SYSTEM ASM_MVCDR (* Assembly System Control+Diagnostics+HMI with Remote Model+View *)
  (* Standard: 61499-1; Classification: Simulation; ApplicationDomain: Assembly; Type: Dual Stroke Cylinder *)
  (* Version 1.0, 2007-11-08, JHC, Holobloc Inc, Changed PRESS_ACT socket from 1027 to 1031. *)
  (* Version 0.9, 2007-07-07, JHC, Holobloc Inc, Added DIAGNOSTICS.LOG.RUN. *)
  (* Version 0.8, 2007-07-07, JHC, Holobloc Inc, Accelerated simulation, adjusted diagnostics; added ASM_GATE to TRANSPORT_MDL, PRESS_MDL. *)
  (* Version 0.7, 2007-07-06, JHC, Holobloc Inc, Simplified MODEL.CLOCK as in ASM_MVCDL. *)
  (* Version 0.6, 2007-07-06, JHC, Holobloc Inc, Added initial readout of TRANSPORT_ACT, PRESS_ACT. *)
  (* Version 0.5, 2007-07-06, JHC, Holobloc Inc, Adjusted order of resources so timing-sensitive initialization is always done last. *)
  (* Version 0.4, 2007-07-05, JHC, Holobloc Inc, Made device order MODEL, DIAGNOSTICS, CONTROL (startup is reverse order). *)
  (* Version 0.3, 2007-07-03, JHC, Holobloc Inc, Updated MODEL.CLOCK as in ASM_MVCL. *)
  (* Version 0.2, 2007-01-15, JHC, Holobloc Inc, Converted I/O to tagged data. *)
  (* Version 0.1, 2004-10-21, JHC, Rockwell Automation, Adapted to new Load/Unload model. *)
  (* Version 0.0, 2004-09-26, JHC, Rockwell Automation, Extended from ASM_MVCDL1. *)
  DEVICE MODEL : RMT_FRAME(BOUNDS := [380,100,185,160])
    RESOURCE MGR : RMT_RES
    END_RESOURCE
    RESOURCE CLOCK : EMB_RES
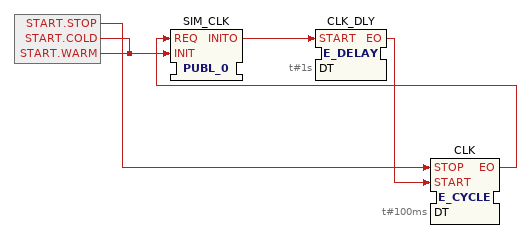
      FBS
        CLK : E_CYCLE(DT := t#100ms);
        SIM_CLK : PUBL_0;
        CLK_DLY : E_DELAY(DT := t#1s); (* Wait for everything to initialize, then start simulation *)
      END_FBS
      EVENT_CONNECTIONS
        CLK.EO TO SIM_CLK.REQ;
        START.STOP TO CLK.STOP;
        START.COLD TO SIM_CLK.INIT;
        START.WARM TO SIM_CLK.INIT;
        SIM_CLK.INITO TO CLK_DLY.START;
        CLK_DLY.EO TO CLK.START;
      END_CONNECTIONS
    END_RESOURCE
    RESOURCE TAGS : EMB_RES
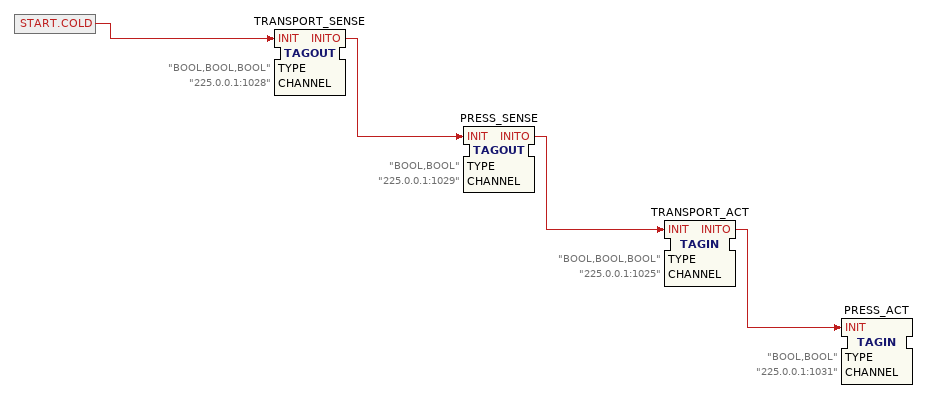
      FBS
        TRANSPORT_SENSE : TAGOUT(TYPE := "BOOL,BOOL,BOOL", CHANNEL := "225.0.0.1:1028");
        TRANSPORT_ACT : TAGIN(TYPE := "BOOL,BOOL,BOOL", CHANNEL := "225.0.0.1:1025");
        PRESS_SENSE : TAGOUT(TYPE := "BOOL,BOOL", CHANNEL := "225.0.0.1:1029");
        PRESS_ACT : TAGIN(TYPE := "BOOL,BOOL", CHANNEL := "225.0.0.1:1031");
      END_FBS
      EVENT_CONNECTIONS
        START.COLD TO TRANSPORT_SENSE.INIT;
        TRANSPORT_ACT.INITO TO PRESS_ACT.INIT;
        TRANSPORT_SENSE.INITO TO PRESS_SENSE.INIT;
        PRESS_SENSE.INITO TO TRANSPORT_ACT.INIT;
      END_CONNECTIONS
    END_RESOURCE
    RESOURCE TRANSPORT_MDL : EMB_RES
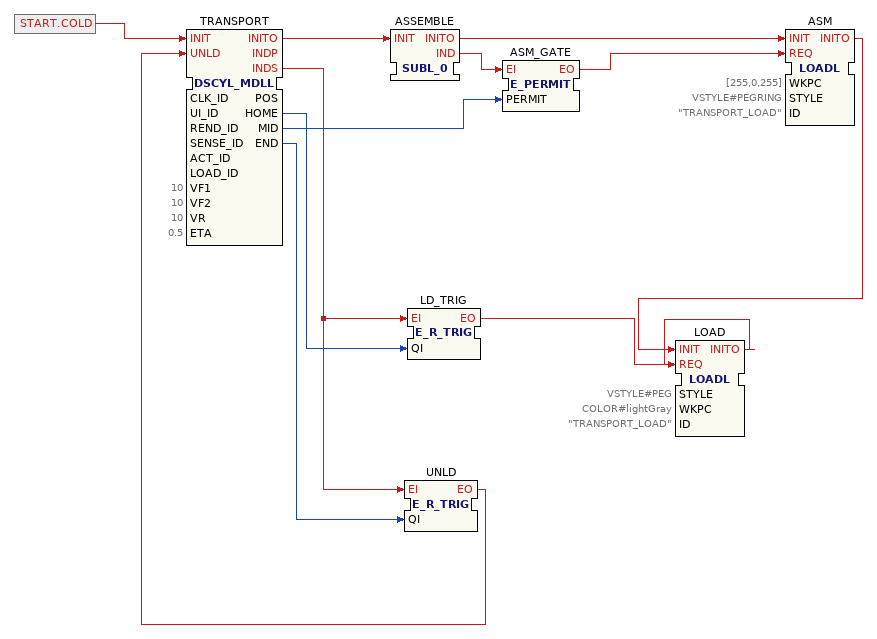
      FBS
        TRANSPORT : DSCYL_MDLL(VF1 := 10, VF2 := 10, VR := 10, ETA := 0.5);
        UNLD : E_R_TRIG;
        ASM : LOADL(WKPC := [255,0,255], STYLE := VSTYLE#PEGRING, ID := "TRANSPORT_LOAD");
        LD_TRIG : E_R_TRIG;
        ASSEMBLE : SUBL_0;
        LOAD : LOADL(STYLE := VSTYLE#PEG, WKPC := COLOR#lightGray, ID := "TRANSPORT_LOAD");
        ASM_GATE : E_PERMIT;
      END_FBS
      EVENT_CONNECTIONS
        TRANSPORT.INDS TO UNLD.EI;
        TRANSPORT.INDS TO LD_TRIG.EI;
        START.COLD TO TRANSPORT.INIT;
        TRANSPORT.INITO TO ASSEMBLE.INIT;
        ASSEMBLE.INITO TO ASM.INIT;
        UNLD.EO TO TRANSPORT.UNLD;
        ASM.INITO TO LOAD.INIT;
        LOAD.INITO TO LOAD.REQ;
        LD_TRIG.EO TO LOAD.REQ;
        ASSEMBLE.IND TO ASM_GATE.EI;
        ASM_GATE.EO TO ASM.REQ;
      END_CONNECTIONS
      DATA_CONNECTIONS
        TRANSPORT.END TO UNLD.QI;
        TRANSPORT.HOME TO LD_TRIG.QI;
        TRANSPORT.MID TO ASM_GATE.PERMIT;
      END_CONNECTIONS
    END_RESOURCE
    RESOURCE PRESS_MDL : EMB_RES
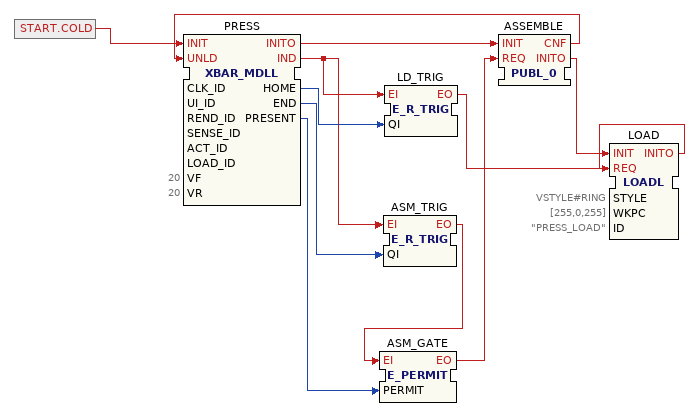
      FBS
        PRESS : XBAR_MDLL(VF := 20, VR := 20);
        ASM_TRIG : E_R_TRIG; (* Gate for assembly event *)
        ASSEMBLE : PUBL_0;
        LD_TRIG : E_R_TRIG;
        LOAD : LOADL(STYLE := VSTYLE#RING, WKPC := [255,0,255], ID := "PRESS_LOAD");
        ASM_GATE : E_PERMIT; (* Do not assemble if no ring present *)
      END_FBS
      EVENT_CONNECTIONS
        START.COLD TO PRESS.INIT;
        PRESS.IND TO LD_TRIG.EI;
        PRESS.IND TO ASM_TRIG.EI;
        PRESS.INITO TO ASSEMBLE.INIT;
        ASSEMBLE.CNF TO PRESS.UNLD;
        ASSEMBLE.INITO TO LOAD.INIT;
        LD_TRIG.EO TO LOAD.REQ;
        LOAD.INITO TO LOAD.REQ;
        ASM_TRIG.EO TO ASM_GATE.EI;
        ASM_GATE.EO TO ASSEMBLE.REQ;
      END_CONNECTIONS
      DATA_CONNECTIONS
        PRESS.END TO ASM_TRIG.QI;
        PRESS.HOME TO LD_TRIG.QI;
        PRESS.PRESENT TO ASM_GATE.PERMIT;
      END_CONNECTIONS
    END_RESOURCE
    RESOURCE ASSEMBLY : VIEW_PANEL(DIA := 25, SIZE := [7,5], VERTICAL := 0)
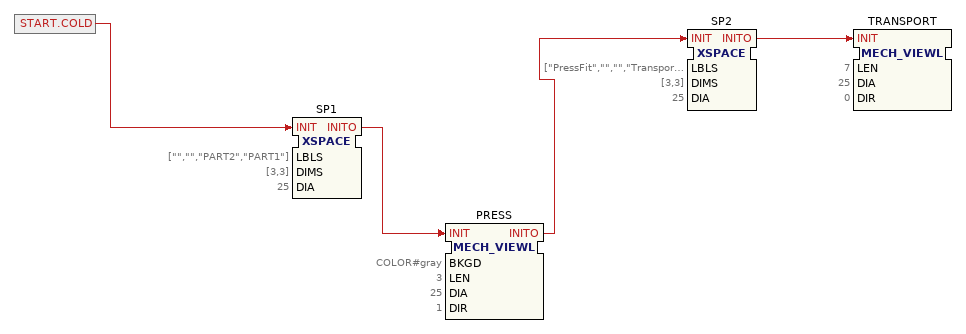
      FBS
        SP1 : XSPACE(LBLS := ["","","PART2","PART1"], DIMS := [3,3], DIA := 25);
        PRESS : MECH_VIEWL(BKGD := COLOR#gray, LEN := 3, DIA := 25, DIR := 1); (* Vertical press element *)
        SP2 : XSPACE(LBLS := ["PressFit","","","Transport"], DIMS := [3,3], DIA := 25);
        TRANSPORT : MECH_VIEWL(LEN := 7, DIA := 25, DIR := 0); (* Dual-Cylinder Transport Mechanism *)
      END_FBS
      EVENT_CONNECTIONS
        START.COLD TO SP1.INIT;
        SP1.INITO TO PRESS.INIT;
        PRESS.INITO TO SP2.INIT;
        SP2.INITO TO TRANSPORT.INIT;
      END_CONNECTIONS
    END_RESOURCE
  END_DEVICE
  DEVICE DIAGNOSTICS : FRAME_DEVICE(BOUNDS := [100,260,465,150], GRID := [1,1])
    RESOURCE TAGS : EMB_RES
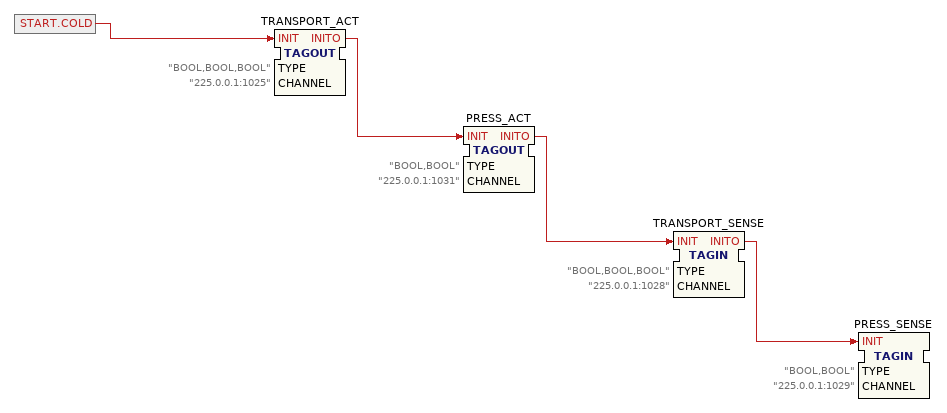
      FBS
        TRANSPORT_SENSE : TAGIN(TYPE := "BOOL,BOOL,BOOL", CHANNEL := "225.0.0.1:1028");
        TRANSPORT_ACT : TAGOUT(TYPE := "BOOL,BOOL,BOOL", CHANNEL := "225.0.0.1:1025");
        PRESS_ACT : TAGOUT(TYPE := "BOOL,BOOL", CHANNEL := "225.0.0.1:1031");
        PRESS_SENSE : TAGIN(TYPE := "BOOL,BOOL", CHANNEL := "225.0.0.1:1029");
      END_FBS
      EVENT_CONNECTIONS
        START.COLD TO TRANSPORT_ACT.INIT;
        TRANSPORT_SENSE.INITO TO PRESS_SENSE.INIT;
        TRANSPORT_ACT.INITO TO PRESS_ACT.INIT;
        PRESS_ACT.INITO TO TRANSPORT_SENSE.INIT;
      END_CONNECTIONS
    END_RESOURCE
    RESOURCE MONITOR : EMB_RES
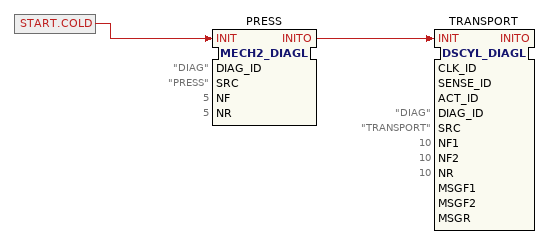
      FBS
        PRESS : MECH2_DIAGL(DIAG_ID := "DIAG", SRC := "PRESS", NF := 5, NR := 5);
        TRANSPORT : DSCYL_DIAGL(DIAG_ID := "DIAG", SRC := "TRANSPORT", NF1 := 10, NF2 := 10, NR := 10);
      END_FBS
      EVENT_CONNECTIONS
        START.COLD TO PRESS.INIT;
        PRESS.INITO TO TRANSPORT.INIT;
      END_CONNECTIONS
    END_RESOURCE
    RESOURCE LOG : PANEL_RESOURCE(ROWS := 1, COLS := 1)
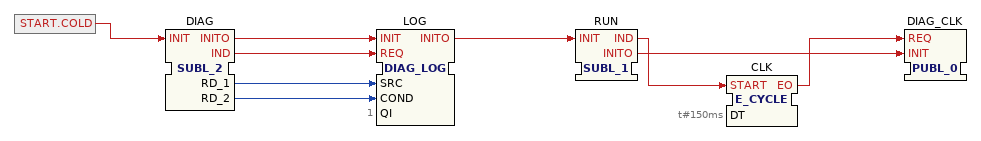
      FBS
        DIAG : SUBL_2;
        LOG : DIAG_LOG(QI := 1);
        CLK : E_CYCLE(DT := t#150ms);
        DIAG_CLK : PUBL_0;
        RUN : SUBL_1;
      END_FBS
      EVENT_CONNECTIONS
        START.COLD TO DIAG.INIT;
        DIAG.INITO TO LOG.INIT;
        DIAG.IND TO LOG.REQ;
        CLK.EO TO DIAG_CLK.REQ;
        LOG.INITO TO RUN.INIT;
        RUN.IND TO CLK.START;
        RUN.INITO TO DIAG_CLK.INIT;
      END_CONNECTIONS
      DATA_CONNECTIONS
        DIAG.RD_1 TO LOG.SRC;
        DIAG.RD_2 TO LOG.COND;
      END_CONNECTIONS
    END_RESOURCE
  END_DEVICE
  DEVICE CONTROL : FRAME_DEVICE(BOUNDS := [100,100,280,160], GRID := [2,2])
    RESOURCE ASSY_CTL : EMB_RES
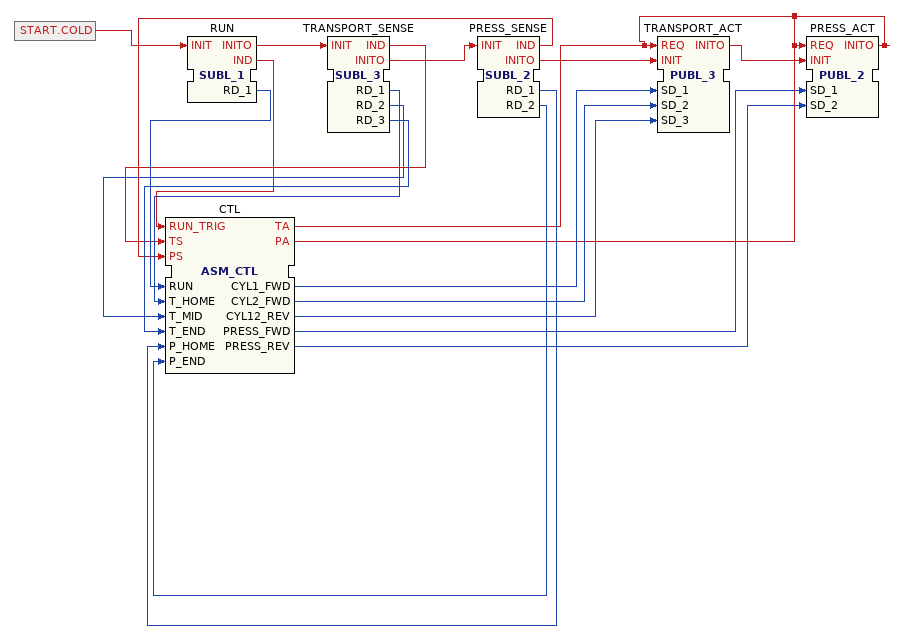
      FBS
        TRANSPORT_SENSE : SUBL_3;
        PRESS_SENSE : SUBL_2;
        TRANSPORT_ACT : PUBL_3;
        PRESS_ACT : PUBL_2;
        CTL : ASM_CTL;
        RUN : SUBL_1;
      END_FBS
      EVENT_CONNECTIONS
        TRANSPORT_SENSE.IND TO CTL.TS;
        CTL.TA TO TRANSPORT_ACT.REQ;
        CTL.PA TO PRESS_ACT.REQ;
        START.COLD TO RUN.INIT;
        RUN.INITO TO TRANSPORT_SENSE.INIT;
        RUN.IND TO CTL.RUN_TRIG;
        TRANSPORT_SENSE.INITO TO PRESS_SENSE.INIT;
        PRESS_SENSE.IND TO CTL.PS;
        PRESS_SENSE.INITO TO TRANSPORT_ACT.INIT;
        TRANSPORT_ACT.INITO TO PRESS_ACT.INIT;
        PRESS_ACT.INITO TO TRANSPORT_ACT.REQ;
        PRESS_ACT.INITO TO PRESS_ACT.REQ;
      END_CONNECTIONS
      DATA_CONNECTIONS
        CTL.CYL1_FWD TO TRANSPORT_ACT.SD_1;
        CTL.CYL2_FWD TO TRANSPORT_ACT.SD_2;
        CTL.CYL12_REV TO TRANSPORT_ACT.SD_3;
        CTL.PRESS_FWD TO PRESS_ACT.SD_1;
        CTL.PRESS_REV TO PRESS_ACT.SD_2;
        TRANSPORT_SENSE.RD_1 TO CTL.T_HOME;
        TRANSPORT_SENSE.RD_2 TO CTL.T_MID;
        TRANSPORT_SENSE.RD_3 TO CTL.T_END;
        PRESS_SENSE.RD_1 TO CTL.P_HOME;
        PRESS_SENSE.RD_2 TO CTL.P_END;
        RUN.RD_1 TO CTL.RUN;
      END_CONNECTIONS
    END_RESOURCE
    RESOURCE TRANSPORT_SENSORS : PANEL_RESOURCE(ROWS := 3, COLS := 1)
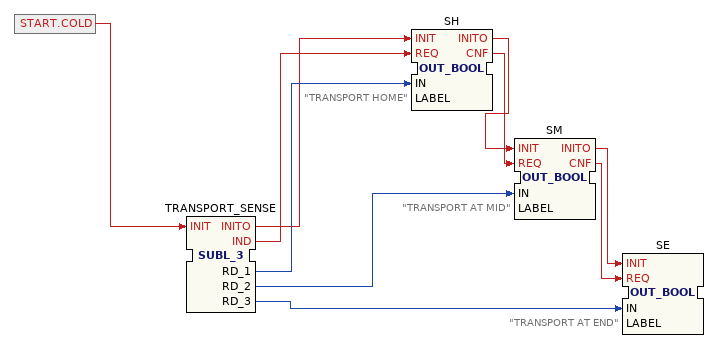
      FBS
        TRANSPORT_SENSE : SUBL_3;
        SH : OUT_BOOL(LABEL := "TRANSPORT HOME");
        SM : OUT_BOOL(LABEL := "TRANSPORT AT MID");
        SE : OUT_BOOL(LABEL := "TRANSPORT AT END");
      END_FBS
      EVENT_CONNECTIONS
        START.COLD TO TRANSPORT_SENSE.INIT;
        TRANSPORT_SENSE.INITO TO SH.INIT;
        SH.INITO TO SM.INIT;
        SM.INITO TO SE.INIT;
        TRANSPORT_SENSE.IND TO SH.REQ;
        SH.CNF TO SM.REQ;
        SM.CNF TO SE.REQ;
      END_CONNECTIONS
      DATA_CONNECTIONS
        TRANSPORT_SENSE.RD_1 TO SH.IN;
        TRANSPORT_SENSE.RD_2 TO SM.IN;
        TRANSPORT_SENSE.RD_3 TO SE.IN;
      END_CONNECTIONS
    END_RESOURCE
    RESOURCE TRANSPORT_ACTUATORS : PANEL_RESOURCE(ROWS := 3, COLS := 1)
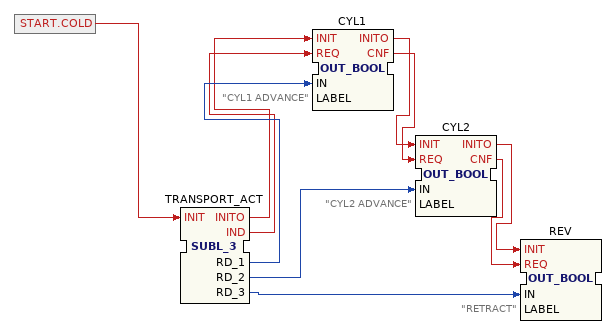
      FBS
        CYL1 : OUT_BOOL(LABEL := "CYL1 ADVANCE");
        CYL2 : OUT_BOOL(LABEL := "CYL2 ADVANCE");
        REV : OUT_BOOL(LABEL := "RETRACT");
        TRANSPORT_ACT : SUBL_3;
      END_FBS
      EVENT_CONNECTIONS
        CYL1.INITO TO CYL2.INIT;
        CYL2.INITO TO REV.INIT;
        CYL2.CNF TO REV.REQ;
        CYL1.CNF TO CYL2.REQ;
        START.COLD TO TRANSPORT_ACT.INIT;
        TRANSPORT_ACT.INITO TO CYL1.INIT;
        TRANSPORT_ACT.IND TO CYL1.REQ;
      END_CONNECTIONS
      DATA_CONNECTIONS
        TRANSPORT_ACT.RD_1 TO CYL1.IN;
        TRANSPORT_ACT.RD_2 TO CYL2.IN;
        TRANSPORT_ACT.RD_3 TO REV.IN;
      END_CONNECTIONS
    END_RESOURCE
    RESOURCE PRESS_SENSORS : PANEL_RESOURCE
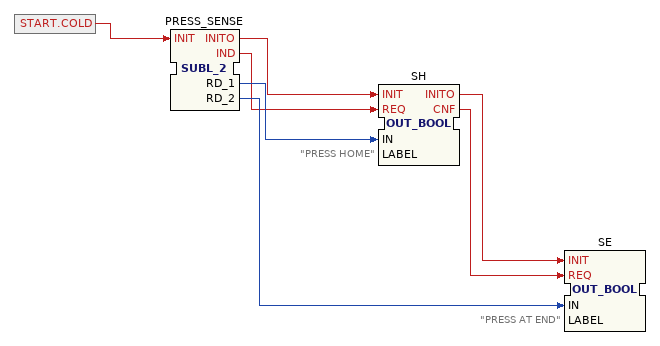
      FBS
        PRESS_SENSE : SUBL_2;
        SH : OUT_BOOL(LABEL := "PRESS HOME");
        SE : OUT_BOOL(LABEL := "PRESS AT END");
      END_FBS
      EVENT_CONNECTIONS
        START.COLD TO PRESS_SENSE.INIT;
        PRESS_SENSE.INITO TO SH.INIT;
        SH.INITO TO SE.INIT;
        PRESS_SENSE.IND TO SH.REQ;
        SH.CNF TO SE.REQ;
      END_CONNECTIONS
      DATA_CONNECTIONS
        PRESS_SENSE.RD_1 TO SH.IN;
        PRESS_SENSE.RD_2 TO SE.IN;
      END_CONNECTIONS
    END_RESOURCE
    RESOURCE PRESS_ACTUATORS : PANEL_RESOURCE
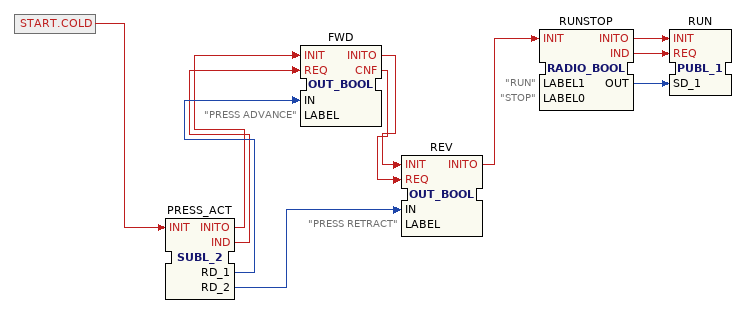
      FBS
        FWD : OUT_BOOL(LABEL := "PRESS ADVANCE");
        REV : OUT_BOOL(LABEL := "PRESS RETRACT");
        PRESS_ACT : SUBL_2;
        RUNSTOP : RADIO_BOOL(LABEL1 := "RUN", LABEL0 := "STOP");
        RUN : PUBL_1;
      END_FBS
      EVENT_CONNECTIONS
        FWD.INITO TO REV.INIT;
        FWD.CNF TO REV.REQ;
        START.COLD TO PRESS_ACT.INIT;
        PRESS_ACT.INITO TO FWD.INIT;
        PRESS_ACT.IND TO FWD.REQ;
        REV.INITO TO RUNSTOP.INIT;
        RUNSTOP.INITO TO RUN.INIT;
        RUNSTOP.IND TO RUN.REQ;
      END_CONNECTIONS
      DATA_CONNECTIONS
        PRESS_ACT.RD_1 TO FWD.IN;
        PRESS_ACT.RD_2 TO REV.IN;
        RUNSTOP.OUT TO RUN.SD_1;
      END_CONNECTIONS
    END_RESOURCE
  END_DEVICE
END_SYSTEM
